{attribute 'enable_dynamic_creation'}
FUNCTION_BLOCK SumCollectorLINT EXTENDS Object IMPLEMENTS ISumCollectorLINT
VAR
	isEnabled :BOOL := TRUE;
	myValue :LINT := 0;
END_VAR

METHOD addValue
VAR_INPUT
	value	: LINT;
END_VAR
RETURN (NOT THIS^.enabled);
THIS^.myValue := THIS^.myValue + value;
END_METHOD

(*

short summary
=================
This abstract property returns the class name of the concrete object, 
which is useful for logging/debugging purpose or to check the class name
for ``__DELETE`` in factories (sometimes it's necessary to do more 
than just to free the memory).

.. <legal notes>

legal notes
=================
| SPDX-FileCopyrightText: © 2022 ekvip automation GmbH <info@ekvip.de>
| SPDX-License-Identifier: Apache-2.0
| For details check: Apache-2.0_

.. _Apache-2.0: https://www.apache.org/licenses/LICENSE-2.0

.. </legal notes>

*)
PROPERTY className : CNM_AbstractObject.ClassName
GET
className := 'SumCollectorLINT';
END_GET
END_PROPERTY

PROPERTY enabled : BOOL
GET
enabled := THIS^.isEnabled;
END_GET
SET
THIS^.isEnabled := enabled;
END_SET
END_PROPERTY

{warning 'Add property implementation'}
PROPERTY sum : LINT
GET
sum := THIS^.myValue;
END_GET
SET
THIS^.myValue := sum;
END_SET
END_PROPERTY

END_FUNCTION_BLOCK

(* stored: Version 1.1.0.1
   POU SumCollectorLINT: Id {a5bcfd4a-6961-425e-8926-a633051e1e1e}, SpecialFunc None
   Method addValue: Id {77bf7b2d-9759-4ada-b5ef-077a5c5ccc3e}
   Property className: Id {a10ac7cf-7639-4fc5-9030-318cf98d2366}
   Get Get: Id {9c0f0154-b545-4405-90e2-5dee253fd021}
   Property enabled: Id {874b888c-b369-421f-bec7-c136045fe68a}
   Get Get: Id {2ed4ff11-968d-43ce-b3d5-02c0191f00b0}
   Set Set: Id {831e23bc-6c64-4091-bb0b-1736a3f2d4ea}
   Property sum: Id {6a20d161-854d-4648-b75d-b7d8cf03a2c4}
   Get Get: Id {877c739a-06cd-43b3-928d-d369325275cd}
   Set Set: Id {8bb68aa1-cff7-41d7-823a-823d330adf2f} *)
